(* IEC 61131-3 sources: learning-path/04_introduction_to_st/src/Namespace, 2 files *)

(* ---- NamespaceExample.st ---- *)
NAMESPACE Circle
    FUNCTION Area : LREAL
        VAR_INPUT
            diameter : LREAL;
        END_VAR
        VAR CONSTANT
            PI : REAL := REAL#3.141592;
        END_VAR
        Area := diameter ** 2.0 * PI / 4.0; // (d^2*PI)/4;
    END_FUNCTION
END_NAMESPACE

NAMESPACE Square
    FUNCTION Area : LREAL
        VAR_INPUT
            sideLength : LREAL;
        END_VAR
        Area := sideLength ** 2.0;
    END_FUNCTION
END_NAMESPACE

(* ---- UsageOfNameSpace.st ---- *)
FUNCTION Calculate : LREAL
    VAR_TEMP
        result : LREAL;
    END_VAR
    result := Circle.Area(diameter := 2.0);    // full qualified call
    result := Square.Area(sideLength := 2.0);  // full qualified call
    ;
END_FUNCTION
